FUNCTION_BLOCK FB_buffer_tote EXTENDS FB_Generic
VAR_INPUT
END_VAR
VAR_OUTPUT
END_VAR
VAR

	fb_rollers		: ARRAY[0..iHas_rollers] OF FB_roller_tote;
	sensor_start	: ARRAY[0..1] OF FB_DigitalInput;//sensor at the beginning of roller[0]
	EDM_24v	: BOOL;//edm_24v
	EDM_sto	: BOOL;//edm_sto
	xError	: BOOL;
	
	
	event				: ST_EVENT;
	rt_error			: R_TRIG;
	bStopped			: BOOL;
	stSubModuleInfo		: ARRAY [1..iSubModule] OF ST_PMLSubUnitInfo;	//Informations about the Subunits
	aUnitInfo	: ARRAY[0..3] OF ST_UnitInfo;
	bMachineStartedUp	: BOOL;
END_VAR
VAR CONSTANT
	iHas_rollers	: INT:=3;
	iSubModule		: UDINT:=4;
	sComponent_name			: STRING := 'fb_buffer';
END_VAR

SUPER^();
IF sensor_start[0].Q OR sensor_start[1].Q THEN
	fb_rollers[0].pre_tote_status := ToteStatus.READY;
ELSE
	fb_rollers[0].pre_tote_status := ToteStatus.EMPTY;
END_IF
fb_rollers[0](	eModeCommand:=eModeCommand,
				eCommand:=eCommand,
				eMode	=>,
				eState =>stSubModuleInfo[1].eState,
				id_roller := 0,
				next_tote_status := fb_rollers[1].current_tote_status
				);
stSubModuleInfo[1].Active			:= TRUE;
fb_rollers[1](	eModeCommand:=eModeCommand,
				eCommand:=eCommand,
				eMode	=>,
				eState =>stSubModuleInfo[2].eState,
				id_roller := 1,
				pre_tote_status := fb_rollers[0].current_tote_status,
				next_tote_status := fb_rollers[2].current_tote_status
				);
stSubModuleInfo[2].Active			:= TRUE;
fb_rollers[2](	eModeCommand:=eModeCommand,
				eCommand:=eCommand,
				eMode	=>,
				eState =>stSubModuleInfo[3].eState,
				id_roller := 2,
				pre_tote_status := fb_rollers[1].current_tote_status,
				next_tote_status := fb_rollers[3].current_tote_status
				);
stSubModuleInfo[3].Active			:= TRUE;
fb_rollers[3](	eModeCommand:=eModeCommand,
				eCommand:=eCommand,
				eMode	=>,
				eState =>stSubModuleInfo[4].eState,
				id_roller := 3,
				pre_tote_status := fb_rollers[2].current_tote_status,
				
				);
stSubModuleInfo[4].Active			:= TRUE;

IF  fb_rollers[0].bUndefinedDone AND fb_rollers[1].bUndefinedDone AND fb_rollers[2].bUndefinedDone AND fb_rollers[3].bUndefinedDone THEN
	bUndefinedDone := TRUE;
END_IF

IF bUndefinedDone AND NOT bMachineStartedUp THEN
	eCommand	:= ePMLCommand_Abort;
	bMachineStartedUp			:= TRUE;
END_IF
//The fbStateMachine from FB_Machine gets the Information about the states and activity from the subunits
fbStateMachine.stSubUnitInfoRef.ArraySize		:= SIZEOF(stSubModuleInfo);
fbStateMachine.stSubUnitInfoRef.NoOfSubUnits	:= iSubModule;
fbStateMachine.stSubUnitInfoRef.pArray			:= ADR(stSubModuleInfo);



//Set unit information 
M_SetUnitInfo();

{attribute 'object_name' := 'M_Aborting'}
METHOD M_Aborting
CASE fbUnitModeManager.eModeStatus OF	
	ePMLProtUnitMode_Production, ePMLProtUnitMode_Manual:		
		G_HMI.bAging_buffer	:= FALSE;
		M_StateComplete();
			
	ePMLProtUnitMode_Maintenance, ePMLUnitMode_Service:
		
		M_StateComplete();
END_CASE
END_METHOD

METHOD M_agingTest : BOOL
VAR_INPUT
END_VAR
FOR i:=0 TO iHas_rollers DO
	fb_rollers[i].M_agingTest();
END_FOR
END_METHOD

{attribute 'object_name' := 'M_Execute'}
METHOD M_Execute

VAR

END_VAR
CASE fbUnitModeManager.eModeStatus OF
	ePMLProtUnitMode_Production:		//Mode Production
		//Processing automatic Seperation
//		IF sensor_start[0].Q OR sensor_start[1].Q THEN
//			fb_rollers[0].pre_tote_status := ToteStatus.READY;
//		ELSE
//			fb_rollers[0].pre_tote_status := ToteStatus.EMPTY;
//		END_IF
//		fb_rollers[0](	id_roller := 0,
//						next_tote_status := fb_rollers[1].current_tote_status);
//		fb_rollers[1](	id_roller := 1,
//						pre_tote_status := fb_rollers[0].current_tote_status,
//						next_tote_status := fb_rollers[2].current_tote_status);
//		fb_rollers[2](	id_roller := 2,
//						pre_tote_status := fb_rollers[1].current_tote_status,
//						next_tote_status := fb_rollers[3].current_tote_status);
//		fb_rollers[3](	id_roller := 3,
//						pre_tote_status := fb_rollers[2].current_tote_status,
//						next_tote_status := GVL.fb_loading.current_tote_status);		
		
	ePMLProtUnitMode_Maintenance, ePMLUnitMode_Service:		
		//
		
	ePMLProtUnitMode_Manual:		//Manaul

END_CASE
END_METHOD

{attribute 'object_name' := 'M_Idle'}
METHOD M_Idle
IF G_HMI.bAging_buffer THEN
	M_agingTest();
END_IF
END_METHOD

METHOD M_mapping : BOOL
VAR_INPUT
END_VAR

//todo:reconfig dios
/////////////////////////////////////digital input////////////////////////////////////////

fb_rollers[0].roller.err			:= G_IO.arDI[1].Ch[0];
fb_rollers[1].roller.err			:= G_IO.arDI[1].Ch[1];
fb_rollers[1].roller.sensor(D:= G_IO.arDI[1].Ch[2],on_ms:=100,off_ms:=100);
fb_rollers[2].roller.sensor(D:= G_IO.arDI[1].Ch[3],on_ms:=100,off_ms:=100);
fb_rollers[2].roller.err			:= G_IO.arDI[1].Ch[4];
fb_rollers[3].roller.err			:= G_IO.arDI[1].Ch[5];
fb_rollers[3].roller.sensor(D:= G_IO.arDI[1].Ch[6],on_ms:=100,off_ms:=100);
fb_rollers[3].sensor_mute(D:= G_IO.arDI[1].Ch[7],on_ms:=10,off_ms:=100);
EDM_24v								:= G_IO.arDI[1].Ch[11];
EDM_sto								:= G_IO.arDI[1].Ch[12];
sensor_start[0](D:= G_IO.arDI[1].Ch[13],on_ms:=100,off_ms:=100);
sensor_start[1](D:= G_IO.arDI[1].Ch[15],on_ms:=100,off_ms:=100);
fb_rollers[0].roller.sensor(D:= G_IO.arDI[1].Ch[14],on_ms:=100,off_ms:=100);

/////////////////////////////////////digital output////////////////////////////////////////
G_IO.arDO[1].Ch[0]	:= fb_rollers[2].roller.forward;
G_IO.arDO[1].Ch[1]	:= fb_rollers[2].roller.backward;
G_IO.arDO[1].Ch[2]	:= fb_rollers[0].roller.forward;
G_IO.arDO[1].Ch[3]	:= fb_rollers[0].roller.backward;
G_IO.arDO[1].Ch[4]	:= fb_rollers[1].roller.forward;
G_IO.arDO[1].Ch[5]	:= fb_rollers[1].roller.backward;
G_IO.arDO[1].Ch[6]	:= fb_rollers[3].roller.forward;
G_IO.arDO[1].Ch[7]	:= fb_rollers[3].roller.backward;



/////////////////////////////////////fb rollers////////////////////////////////////////

FOR i:=0 TO iHas_rollers DO
	fb_rollers[i].M_mapping();
END_FOR
END_METHOD

METHOD M_Reset
VAR_INPUT
END_VAR
//Take away all commands
IF GVL.stChangeIntoProduction.bYesReset THEN
;
END_IF
END_METHOD

{attribute 'object_name' := 'M_Resetting'}
METHOD M_Resetting
CASE fbUnitModeManager.eModeStatus OF
	ePMLProtUnitMode_Production:		//Production, Mantainance, Manual	
		M_StateComplete();
	
	ePMLProtUnitMode_Maintenance, ePMLProtUnitMode_Manual, ePMLUnitMode_Service:
		M_StateComplete();
END_CASE
END_METHOD

METHOD M_SetUnitInfo
VAR_INPUT
END_VAR
aUnitInfo[0].Name			:= 'roller[0]';
aUnitInfo[0].ActMode			:= eMode;
aUnitInfo[0].ActState		:= eState;

aUnitInfo[1].Name				:= 'roller[1]';
aUnitInfo[1].ActMode			:= GVL.fb_buffer.eMode;
aUnitInfo[1].ActState			:= GVL.fb_buffer.eState;

aUnitInfo[2].Name			:= 'roller[2]';
aUnitInfo[2].ActMode			:= GVL.fb_buffer.eMode;
aUnitInfo[2].ActState		:= GVL.fb_buffer.eState;

aUnitInfo[3].Name			:= 'roller[3]';
aUnitInfo[3].ActMode			:= GVL.fb_buffer.eMode;
aUnitInfo[3].ActState		:= GVL.fb_buffer.eState;
END_METHOD

{attribute 'object_name' := 'M_Starting'}
METHOD M_Starting
CASE fbUnitModeManager.eModeStatus OF
	ePMLProtUnitMode_Production:		//Production, Mantainance, Manual
		//Resetting all Commands and Values
		G_HMI.bAging_test	:= FALSE;
		M_StateComplete();

	ePMLProtUnitMode_Maintenance, ePMLProtUnitMode_Manual, ePMLUnitMode_Service:
		M_StateComplete();
END_CASE
END_METHOD

{attribute 'object_name' := 'M_Stopping'}
METHOD M_Stopping
CASE fbUnitModeManager.eModeStatus OF
	ePMLProtUnitMode_Production, ePMLProtUnitMode_Manual:			
		M_StateComplete();

	ePMLProtUnitMode_Maintenance, ePMLUnitMode_Service:
		M_StateComplete();	
			//not defined
END_CASE
END_METHOD

{attribute 'object_name' := 'M_Undefined'}
METHOD M_Undefined

bUndefinedDone					:= TRUE;
END_METHOD

END_FUNCTION_BLOCK

(* stored: Version 1.1.0.1, ProductVersion 3.1.4024.12
   POU FB_buffer_tote: Id {19049f21-ed2b-4a13-83c2-eea6536c4f38}, SpecialFunc None
   Method M_Aborting: Id {8bebec9d-60c2-4ac7-bf32-efe186b9bfd8}
   Method M_agingTest: Id {005eedab-3965-4f90-9be8-7f9d4d5a9fec}
   Method M_Execute: Id {6c772562-34c8-47b4-91c2-3dd9e3a0282e}
   Method M_Idle: Id {852a977a-fb07-4f73-b57c-37d614c8411c}
   Method M_mapping: Id {1382acc9-2aac-40e5-9b78-e873bc29d4e0}
   Method M_Reset: Id {828769aa-b396-465f-9a50-434ca369865f}
   Method M_Resetting: Id {9a1f29a5-17c7-492c-91f2-093b5dd6c83b}
   Method M_SetUnitInfo: Id {c1d055cf-d164-4699-93b1-6e91a9f5fa94}
   Method M_Starting: Id {dda3e1fd-29c7-41f0-889f-35f057fc9945}
   Method M_Stopping: Id {e0c357c3-0799-40ea-9f63-65c4fab25377}
   Method M_Undefined: Id {9298f8b5-e108-4edf-8894-8f62c357fbb0} *)
